TYPE U_FanucCNCEventInfo :
UNION
	{attribute 'displaymode':='hex'}
	Id : WORD;
	Details : ST_FanucCNCEventDetails;
END_UNION

END_TYPE

(* stored: Version 1.1.0.1, ProductVersion 3.1.4024.12
   DUT U_FanucCNCEventInfo: Id {26cd41bd-47cc-4ec2-9397-8f37ea14bd02} *)
